
(* ===== HMI "Unified PC RT_4" =====

HMI tags "sql"
   "column1" : Array [0..99] of WString[254], internal
   "column2" : Array [0..99] of WString[254], internal
   "column3" : Array [0..99] of WString[254], internal
   "sqlUDT" : c2be0524-ca88-4e16-9980-a7dd9fce2099, internal
   "column5" : Array [0..99] of WString[254], internal
   "column4" : Array [0..99] of WString[254], internal
*)